% RSLogix 500 project I2P HANDS-ON 3 - LUKE.RSS, saved by version 10.00.00.00 %
PROJECT "UNTITLED"    % processor: Bul.1763 MicroLogix 1100 Series B %

PROGRAM FILES
  LAD 2   9 rungs

DATA FILES
  O0 OUTPUT  4 elements
  I1 INPUT  6 elements
  S2 STATUS  66 elements
  B3 BINARY  1 elements
  T4 TIMER  2 elements
  C5 COUNTER  1 elements
  R6 CONTROL  1 elements
  N7 INTEGER  1 elements
  F8 FLOAT  1 elements

LADDER 2
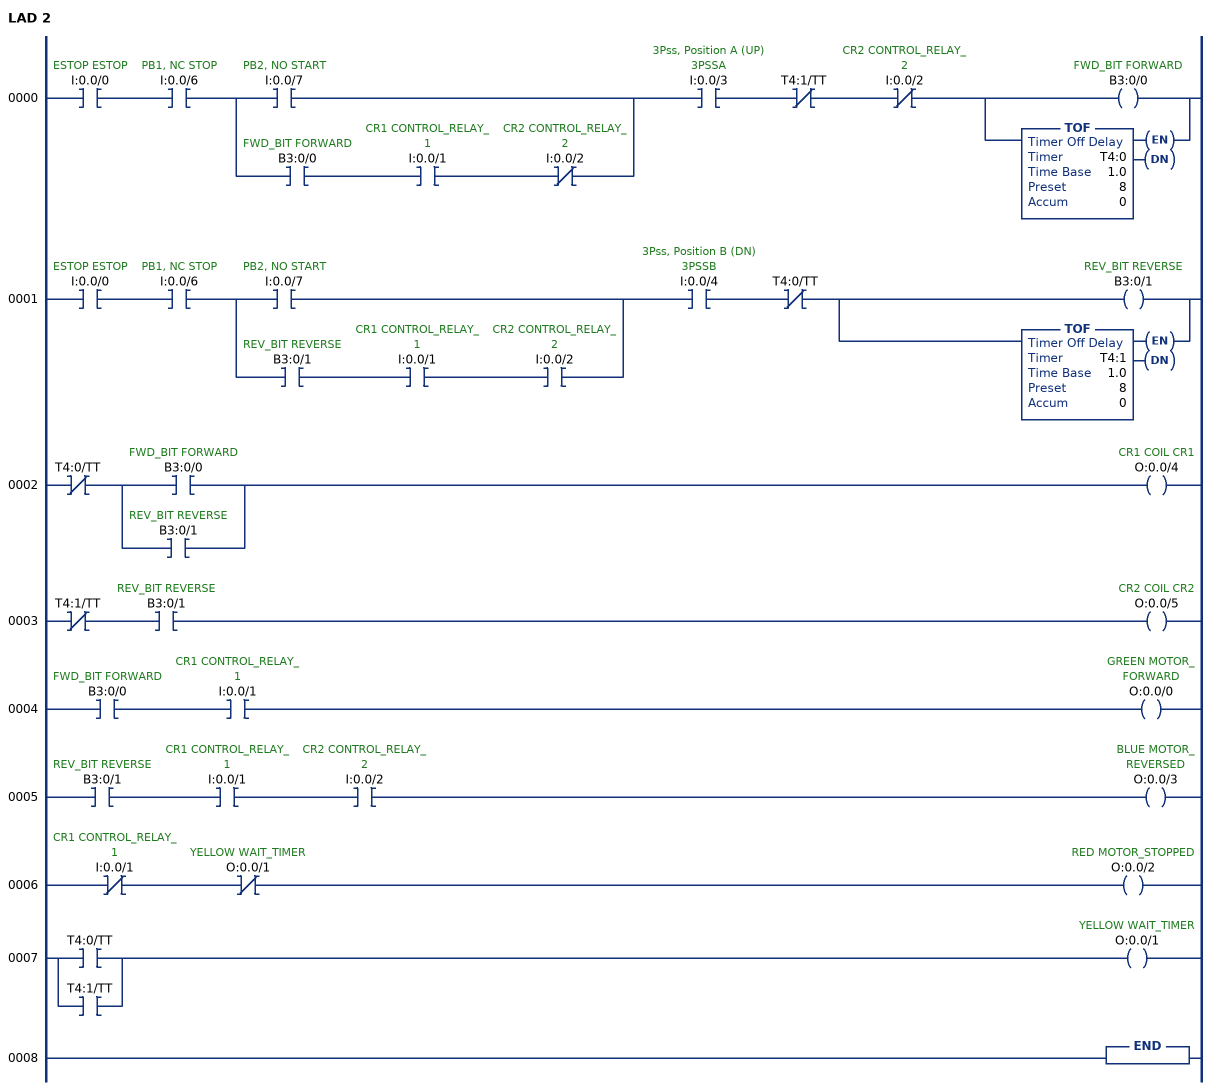
% Rung: 0 %
SOR XIC I:0.0/0 XIC I:0.0/6 BST XIC I:0.0/7 NXB XIC B3:0/0 XIC I:0.0/1 XIO I:0.0/2 BND XIC I:0.0/3 XIO T4:1/TT XIO I:0.0/2 BST OTE B3:0/0 NXB TOF T4:0 1.0 8 0 BND EOR
%   I:0.0/0  ESTOP  "ESTOP" %
%   I:0.0/6  STOP  "PB1, NC" %
%   I:0.0/7  START  "PB2, NO" %
%   B3:0/0  FORWARD  "FWD_BIT" %
%   I:0.0/1  CONTROL_RELAY_1  "CR1" %
%   I:0.0/2  CONTROL_RELAY_2  "CR2" %
%   I:0.0/3  3PSSA  "3Pss, Position A (UP)" %
% Rung: 1 %
SOR XIC I:0.0/0 XIC I:0.0/6 BST XIC I:0.0/7 NXB XIC B3:0/1 XIC I:0.0/1 XIC I:0.0/2 BND XIC I:0.0/4 XIO T4:0/TT BST OTE B3:0/1 NXB TOF T4:1 1.0 8 0 BND EOR
%   I:0.0/0  ESTOP  "ESTOP" %
%   I:0.0/6  STOP  "PB1, NC" %
%   I:0.0/7  START  "PB2, NO" %
%   B3:0/1  REVERSE  "REV_BIT" %
%   I:0.0/1  CONTROL_RELAY_1  "CR1" %
%   I:0.0/2  CONTROL_RELAY_2  "CR2" %
%   I:0.0/4  3PSSB  "3Pss, Position B (DN)" %
% Rung: 2 %
SOR XIO T4:0/TT BST XIC B3:0/0 NXB XIC B3:0/1 BND OTE O:0.0/4 EOR
%   B3:0/0  FORWARD  "FWD_BIT" %
%   B3:0/1  REVERSE  "REV_BIT" %
%   O:0.0/4  CR1  "CR1 COIL" %
% Rung: 3 %
SOR XIO T4:1/TT XIC B3:0/1 OTE O:0.0/5 EOR
%   B3:0/1  REVERSE  "REV_BIT" %
%   O:0.0/5  CR2  "CR2 COIL" %
% Rung: 4 %
SOR XIC B3:0/0 XIC I:0.0/1 OTE O:0.0/0 EOR
%   B3:0/0  FORWARD  "FWD_BIT" %
%   I:0.0/1  CONTROL_RELAY_1  "CR1" %
%   O:0.0/0  MOTOR_FORWARD  "GREEN" %
% Rung: 5 %
SOR XIC B3:0/1 XIC I:0.0/1 XIC I:0.0/2 OTE O:0.0/3 EOR
%   B3:0/1  REVERSE  "REV_BIT" %
%   I:0.0/1  CONTROL_RELAY_1  "CR1" %
%   I:0.0/2  CONTROL_RELAY_2  "CR2" %
%   O:0.0/3  MOTOR_REVERSED  "BLUE" %
% Rung: 6 %
SOR XIO I:0.0/1 XIO O:0.0/1 OTE O:0.0/2 EOR
%   I:0.0/1  CONTROL_RELAY_1  "CR1" %
%   O:0.0/1  WAIT_TIMER  "YELLOW" %
%   O:0.0/2  MOTOR_STOPPED  "RED" %
% Rung: 7 %
SOR BST XIC T4:0/TT NXB XIC T4:1/TT BND OTE O:0.0/1 EOR
%   O:0.0/1  WAIT_TIMER  "YELLOW" %
% Rung: 8 %
SOR END EOR

OTHER DOCUMENTED ADDRESSES
  NOT_YELLOW  "NOT YELLOW"
  TT  "NOT YELLOW"

DATA TABLE (non-zero values as saved)
DATA T4
% .PRE .ACC %
% T4:0 % 8 0
% T4:1 % 8 0
